PROGRAM MAIN
VAR
	bTest : BOOL;
END_VAR

END_PROGRAM

(* stored: Version 1.1.0.1, ProductVersion 3.1.4024.11
   POU MAIN: Id {956534fd-20d9-4764-8e8b-1cc7ffbf3fb8}, SpecialFunc None *)
